TYPE ST_TIME_PROPORTIONAL_THERMOSTAT_STATE :
STRUCT
	on:					BOOL;
	cycleTimeExpired:	TIME;
	calculatedOnTime:	TIME;
END_STRUCT
END_TYPE

(* stored: Version 1.1.0.1
   DUT ST_TIME_PROPORTIONAL_THERMOSTAT_STATE: Id {7c673e0e-a754-4d66-8773-cbd3de165470} *)
